PROGRAM MAIN
VAR
	
	// Establish state machine for hardware
	MASTER_STATE : MasterStateType := MasterStateType.WAITING;
	PREVIOUS_MASTER_STATE : MasterStateType := MasterStateType.WAITING; 
	MASTER_STATE_STR : STRING := TO_STRING(MASTER_STATE);

	// Establish state machine for GUI
	WINDOW_STATE : ActiveWindowStateType := ActiveWindowStateType.EXPERIMENT_WINDOW; 
	
	// Load submodules 
	fbMainExperimentBlock : MainExperimentBlock; 
	
END_VAR

// Update master state string to send to GUI 
MASTER_STATE_STR := TO_STRING(MASTER_STATE);

// Based on the master state, load different behavior profile. 

// Check to make sure that we command the motor to 0 and reset encoder after we're exiting this state 
IF PREVIOUS_MASTER_STATE = MasterStateType.ACTIVE AND MASTER_STATE <> MasterStateType.ACTIVE THEN
	fbMainExperimentBlock.Reset(); 
END_IF

CASE MASTER_STATE OF
	MasterStateType.ACTIVE : fbMainExperimentBlock(); 
	MasterStateType.CALIBRATION : CalibrationExperimentLoop();
END_CASE

// Update previous master state, recall master state 
// itself is controlled by GUI
PREVIOUS_MASTER_STATE := MASTER_STATE;

END_PROGRAM

(* stored: Version 1.1.0.1, ProductVersion 3.1.4024.12
   POU MAIN: Id {b28e76a4-304f-4046-9598-fedbe83adcc0}, SpecialFunc None *)
